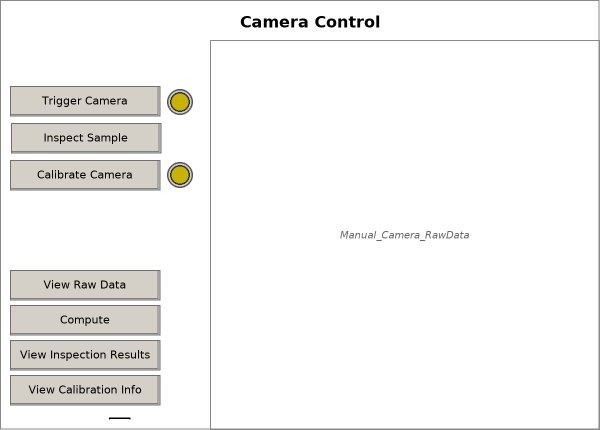
VISUALIZATION Manual_Camera  // 600x430
    Label (133,7 355x30), "Camera Control"
    Button (11,123 150x30), "Inspect Sample", input disabled if: MAIN.fbSlitter.bBusy
        OnMouseClick: execute { MAIN.fbSlitter.Manual.bCameraInspect := TRUE; }
    Button (10,86 150x30), "Trigger Camera", input disabled if: MAIN.fbSlitter.bBusy
        OnMouseClick: execute { MAIN.fbSlitter.Manual.bCameraTrigger := TRUE; }
    Button (10,160 150x30), "Calibrate Camera", input disabled if: MAIN.fbSlitter.bBusy
        OnMouseClick: execute { MAIN.fbSlitter.Manual.bCameraCalibrate := TRUE; }
        OnMouseClick: FrameSelectionChange Selection=SelectedFrame=62eee777-8d81-454f-aaa1-e694c65750cd, Selection=2, GlobSel=AssignType=Directly, SelType=Locally
    Lamp1 (165,87 30x30), variable: MAIN.fbSlitter.Camera.Trigger, style: Lamp-Lamp1-Yellow
    Lamp1 (165,160 30x30), variable: MAIN.fbSlitter.bCalibration, style: Lamp-Lamp1-Yellow
    Frame (210,40 390x390)
        shows Manual_Camera_RawData()
        shows Manual_Camera_Inspection_Raw()
        shows Manual_Camera_Calibration()
        shows Manual_Select_Tube()
    Button (10,270 150x30), "View Raw Data"
        OnMouseClick: FrameSelectionChange Selection=SelectedFrame=62eee777-8d81-454f-aaa1-e694c65750cd, GlobSel=AssignType=Directly, SelType=Locally
        OnMouseClick: execute { MAIN.fbSlitter.Manual.bCameraRawData := TRUE; }
    Button (10,340 150x30), "View Inspection Results"
        OnMouseClick: FrameSelectionChange Selection=SelectedFrame=62eee777-8d81-454f-aaa1-e694c65750cd, Selection=1, GlobSel=AssignType=Directly, SelType=Locally
    Button (10,375 150x30), "View Calibration Info"
        OnMouseClick: FrameSelectionChange Selection=SelectedFrame=62eee777-8d81-454f-aaa1-e694c65750cd, Selection=2, GlobSel=AssignType=Directly, SelType=Locally
    Button (10,305 150x30), "Compute"
        OnMouseClick: execute { Main.fbSlitter.Manual.bCameraComputePeak := TRUE; }
    Rectangle (109,418 21x0)
END_VISUALIZATION

(* stored: Version 1.1.0.1, ProductVersion 3.1.4024.9
   Visu Manual_Camera: Id {6b6210d8-1af0-48a7-ad29-a24cef3564c8} *)
